ABB RobotStudio station: ProyectoLab.rsstn

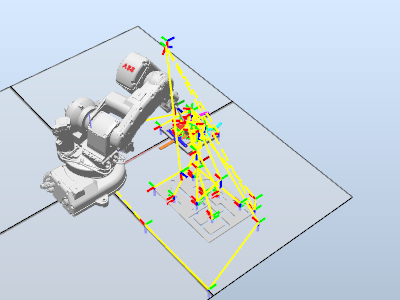
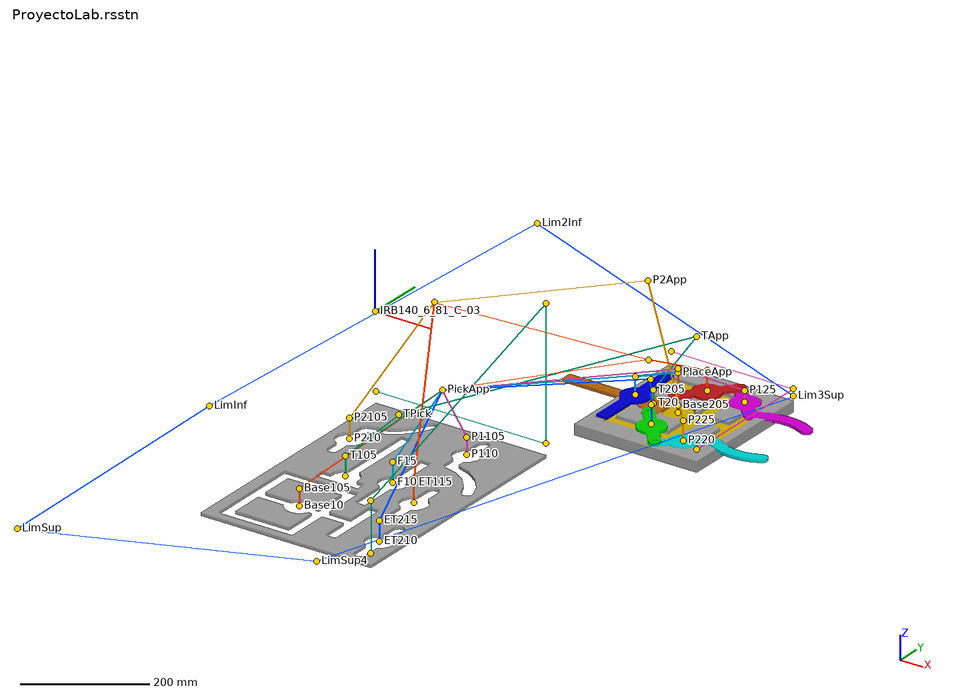
[picture v1: parts stored in the station drawn from their meshes, with robot base, taught points and paths (robot models come from the ABB library and are not in the file)]
Station ProyectoLab (saved by RobotStudio 22.2.9947.0)
Controller ProyectoLab
  mechanical unit ROB_1: IRB140_6_81_C_03, 6 joints, base frame (0, 0, 0) mm
Layout (positions relative to the parent item):
  - IRB140_6_81_C_03 [mechanism, from Robots\IRB140_6_81_C_G_03.rslib] at (0, 0, 0) mm; joint values [0.2279, 1.2634, -0.2779, 1.7688, -1.7005, -0.5808] (rad or m)
  - NewChupa [mechanism] at (606.41, 75.75, 144.2) mm, rotated rx -90 ry 89.52 rz 179.52 deg
      TCP NewChupa at (-10.65, -116.78, 115.87) mm, rotated rx -90 ry 89.52 rz -179.52 deg
      links: Chupita2
  - PiezaACortarApoyoInicialV3_0 [part] at (541.15, -381.68, 0) mm, rotated rx 90 ry 0 rz 180 deg, size 320 x 5 x 470 mm
  - TablaDejarV3 [part] at (639.18, -60.56, -43.75) mm, rotated rx 90 ry 0 rz 180 deg, size 230 x 19 x 260 mm
  - BaseGripper [part] at (583.77, -50.6, 10) mm, rotated rx 90 ry 0 rz 180 deg, size 200 x 5 x 180 mm
  - EslabonTransmisor1 [part] at (606.72, 23.71, 20) mm, rotated rx 90 ry 0 rz -39.33 deg, size 50 x 5 x 124.5 mm
  - EslabonTransmisor2 [part] at (606.64, -124.82, 20) mm, rotated rx 90 ry 0 rz 40 deg, size 50 x 5 x 124.5 mm
  - Pinza1 [part] at (672.04, 32.31, 20) mm, rotated rx -90 ry 0 rz 45 deg, size 111 x 5 x 174 mm
  - Pinza2 [part] at (672.04, -133.51, 15) mm, rotated rx 90 ry 0 rz -45 deg, size 111 x 5 x 174 mm
  - PlacaRetencion [part] at (523.76, -50.61, 20) mm, rotated rx 90 ry 0 rz 0 deg, size 49.7 x 5 x 180 mm
  - T [part] at (573.29, -50.6, 15) mm, rotated rx 90 ry 0 rz 180 deg, size 190 x 5 x 80 mm
  - IniB [smart component, from Components\Positioner.rslib]
      properties: Object=BaseGripper; Position=[0.28101 -0.63451 0]; Orientation=[1.5707963267949 0 3.14159265358979]; Reference=Global; ReferenceObject=(none)
  - IniT [smart component, from Components\Positioner.rslib]
      properties: Object=T; Position=[0.29968 -0.52272 0]; Orientation=[1.5707963267949 0 1.5707963267949]; Reference=Global; ReferenceObject=(none)
  - IniP1 [smart component, from Components\Positioner.rslib]
      properties: Object=Pinza1; Position=[0.40971 -0.3395 0.005]; Orientation=[-1.5707963267949 0 0]; Reference=Global; ReferenceObject=(none)
  - IniP2 [smart component, from Components\Positioner.rslib]
      properties: Object=Pinza2; Position=[0.2292 -0.39631 0]; Orientation=[1.5707963267949 0 0]; Reference=Global; ReferenceObject=(none)
  - IniE1 [smart component, from Components\Positioner.rslib]
      properties: Object=EslabonTransmisor1; Position=[0.43971 -0.52448 0]; Orientation=[1.5707963267949 0 0]; Reference=Global; ReferenceObject=(none)
  - IniE2 [smart component, from Components\Positioner.rslib]
      properties: Object=EslabonTransmisor2; Position=[0.47319 -0.6645 0]; Orientation=[1.5707963267949 0 0]; Reference=Global; ReferenceObject=(none)
  - IniPR [smart component, from Components\Positioner.rslib]
      properties: Object=PlacaRetencion; Position=[0.37233 -0.48425 0]; Orientation=[1.5707963267949 0 0]; Reference=Global; ReferenceObject=(none)
  - finB [smart component, from Components\Positioner.rslib]
      properties: Object=BaseGripper; Position=[0.58377 -0.0506 0.01]; Orientation=[1.5707963267949 0 -3.14159265358979]; Reference=Global; ReferenceObject=(none)
  - finT [smart component, from Components\Positioner.rslib]
      properties: Object=T; Position=[0.57329 -0.0506 0.015]; Orientation=[1.5707963267949 0 3.14159265358979]; Reference=Global; ReferenceObject=(none)
  - finP1 [smart component, from Components\Positioner.rslib]
      properties: Object=Pinza1; Position=[0.67204 0.03231 0.02]; Orientation=[-1.5707963267949 0 0.785398163397448]; Reference=Global; ReferenceObject=(none)
  - finP2 [smart component, from Components\Positioner.rslib]
      properties: Object=Pinza2; Position=[0.67204 -0.13351 0.015]; Orientation=[1.5707963267949 0 -0.785398163397448]; Reference=Global; ReferenceObject=(none)
  - finE1 [smart component, from Components\Positioner.rslib]
      properties: Object=EslabonTransmisor1; Position=[0.60672 0.02371 0.02]; Orientation=[1.5707963267949 0 -0.68643799480937]; Reference=Global; ReferenceObject=(none)
  - finE2 [smart component, from Components\Positioner.rslib]
      properties: Object=EslabonTransmisor2; Position=[0.60664 -0.12482 0.02]; Orientation=[1.5707963267949 0 0.698131700797732]; Reference=Global; ReferenceObject=(none)
  - finPR [smart component, from Components\Positioner.rslib]
      properties: Object=PlacaRetencion; Position=[0.52376 -0.05061 0.02]; Orientation=[1.5707963267949 0 0]; Reference=Global; ReferenceObject=(none)
  - Frame_1 [frame] at (127.2, 0.49, 126.37) mm, rotated rx -90 ry 89.52 rz -89.52 deg
Attachment: NewChupa is attached to IRB140_6_81_C_03 / Link6
Station signals: DI B1, DI B2, DI T1, DI T2, DI P11, DI P12, DI P21, DI P22, DI E11, DI E12, DI E21, DI E22, DI F1, DI F2
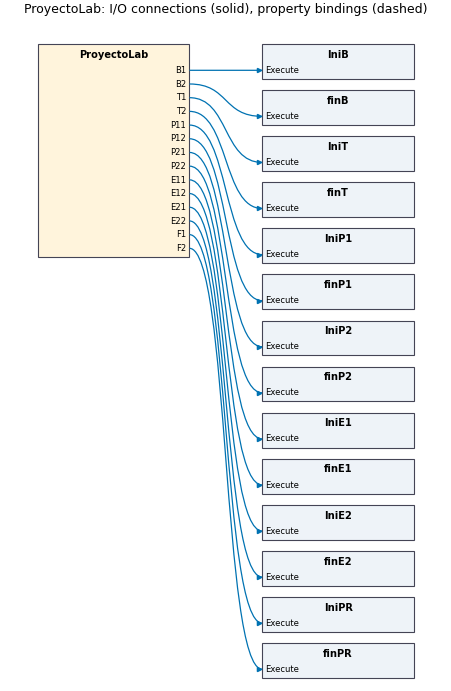
Station logic (signal -> signal, property => property):
  ProyectoLab.B1 -> IniB.Execute
  ProyectoLab.B2 -> finB.Execute
  ProyectoLab.T1 -> IniT.Execute
  ProyectoLab.T2 -> finT.Execute
  ProyectoLab.P11 -> IniP1.Execute
  ProyectoLab.P12 -> finP1.Execute
  ProyectoLab.P21 -> IniP2.Execute
  ProyectoLab.P22 -> finP2.Execute
  ProyectoLab.E11 -> IniE1.Execute
  ProyectoLab.E12 -> finE1.Execute
  ProyectoLab.E21 -> IniE2.Execute
  ProyectoLab.E22 -> finE2.Execute
  ProyectoLab.F1 -> IniPR.Execute
  ProyectoLab.F2 -> finPR.Execute
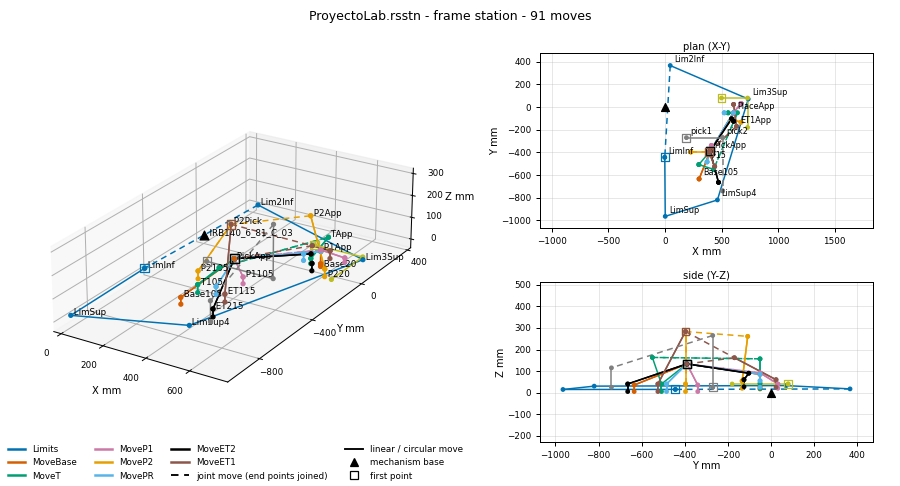
[picture p0: tool path of ProyectoLab.rsstn in frame station, 91 of 98 moves have a stored position in this frame; points joined in program order, loops and branches not executed]
Targets, tools, work objects and paths stored in the station, written as RAPID:
! task T_ROB1
MODULE CalibData
  PERS tooldata NewChupa:=[TRUE,[[127.2,0.485,126.368],[0.707106781,-0.005923775,0.707081968,0]],[1,[83.322,0.242,104.5],[1,0,0,0],0,0,0]];
  TASK PERS wobjdata World:=[FALSE,TRUE,"",[[0,0,0],[1,0,0,0]],[[0,0,0],[1,0,0,0]]];
  TASK PERS wobjdata NewPick:=[FALSE,TRUE,"",[[510,-270,5],[0,1,0,0]],[[0,0,0],[1,0,0,0]]];
  TASK PERS wobjdata NewPlace:=[FALSE,TRUE,"",[[730,80,20],[0,1,0,0]],[[0,0,0],[1,0,0,0]]];
ENDMODULE

! task T_ROB1
MODULE Module1
  CONST robtarget LimInf:=[[-1.268558474,-443.594527115,14.946918722],[0,0.707106781,0.707106781,0],[-1,-2,1,0],[9E+09,9E+09,9E+09,9E+09,9E+09,9E+09]];
  CONST robtarget LimSup:=[[2.920655475,-964.874814922,14.510384672],[0,0.707106781,0.707106781,0],[-1,-2,1,0],[9E+09,9E+09,9E+09,9E+09,9E+09,9E+09]];
  CONST robtarget LimSup4:=[[463.722752628,-820,30.05181616],[0,0.707106781,0.707106781,0],[-1,-2,1,0],[9E+09,9E+09,9E+09,9E+09,9E+09,9E+09]];
  CONST robtarget Lim3Sup:=[[735.880314711,71.133179396,32.548470254],[-0.000000014,0.707106783,0.707106779,0.000000019],[0,-1,1,0],[9E+09,9E+09,9E+09,9E+09,9E+09,9E+09]];
  CONST robtarget Lim2Inf:=[[46.954799307,367.02539237,17.249386066],[0,0.707106781,0.707106781,0],[0,-1,1,0],[9E+09,9E+09,9E+09,9E+09,9E+09,9E+09]];
  CONST robtarget PickApp:=[[-110.342872773,120.113138802,-128.175841477],[0.707106781,0,0,-0.707106781],[-1,0,-1,1],[9E+09,9E+09,9E+09,9E+09,9E+09,9E+09]];
  CONST robtarget Base105:=[[-207.99,364.51,-30],[0.707106781,0,0,-0.707106781],[-1,0,-1,1],[9E+09,9E+09,9E+09,9E+09,9E+09,9E+09]];
  CONST robtarget Base10:=[[-207.99,364.511,0],[0.707106781,0,0,-0.707106781],[-1,0,-1,1],[9E+09,9E+09,9E+09,9E+09,9E+09,9E+09]];
  CONST robtarget PlaceApp:=[[-125.227,130.603,-65],[0.707106781,0,0,-0.707106781],[0,1,-1,1],[9E+09,9E+09,9E+09,9E+09,9E+09,9E+09]];
  CONST robtarget Base205:=[[-125.227,130.604,-8.971],[0.707106781,0,0,-0.707106781],[0,1,-1,1],[9E+09,9E+09,9E+09,9E+09,9E+09,9E+09]];
  CONST robtarget Base20:=[[-125.227,130.604,3],[0.707106781,0,0,-0.707106781],[0,1,-1,1],[9E+09,9E+09,9E+09,9E+09,9E+09,9E+09]];
  CONST robtarget T105:=[[-210.324,237.721,-35],[0.707106781,0,0,-0.707106781],[-1,0,-1,1],[9E+09,9E+09,9E+09,9E+09,9E+09,9E+09]];
  CONST robtarget T10:=[[-210.324,237.721,0],[0.707106781,0,0,-0.707106781],[-1,0,-1,1],[9E+09,9E+09,9E+09,9E+09,9E+09,9E+09]];
  CONST robtarget TPick:=[[-80.342872773,280.113138802,-158.175841477],[0.707106781,0,0,-0.707106781],[-1,0,-1,1],[9E+09,9E+09,9E+09,9E+09,9E+09,9E+09]];
  CONST robtarget TApp:=[[-90.227,130.604,-136.705],[0,0,0,1],[-1,-1,0,1],[9E+09,9E+09,9E+09,9E+09,9E+09,9E+09]];
  CONST robtarget T205:=[[-171.711,130.604,-22.457885204],[0,0,0,1],[-1,-1,-1,1],[9E+09,9E+09,9E+09,9E+09,9E+09,9E+09]];
  CONST robtarget T20:=[[-171.711,130.604,1],[0,0,0,1],[-1,-1,-1,1],[9E+09,9E+09,9E+09,9E+09,9E+09,9E+09]];
  CONST robtarget P1105:=[[-100.292,69.504,-30],[0.707106781,0,0,-0.707106781],[-1,0,-1,1],[9E+09,9E+09,9E+09,9E+09,9E+09,9E+09]];
  CONST robtarget P110:=[[-100.292,69.504,0],[0.707106781,0,0,-0.707106781],[-1,0,-1,1],[9E+09,9E+09,9E+09,9E+09,9E+09,9E+09]];
  CONST robtarget P1App:=[[-125.227,130.604,-71.705],[0.382683433,0,0,-0.923879532],[0,0,-1,1],[9E+09,9E+09,9E+09,9E+09,9E+09,9E+09]];
  CONST robtarget P125:=[[-57.955,47.693,-20],[0.382683433,0,0,-0.923879532],[0,0,-1,1],[9E+09,9E+09,9E+09,9E+09,9E+09,9E+09]];
  CONST robtarget P120:=[[-57.955,47.693,0],[0.382683433,0,0,-0.923879532],[0,0,-1,1],[9E+09,9E+09,9E+09,9E+09,9E+09,9E+09]];
  CONST robtarget P2Pick:=[[-121.178397921,126.307,-278.381942838],[0,0,0,1],[-1,1,-2,0],[9E+09,9E+09,9E+09,9E+09,9E+09,9E+09]];
  CONST robtarget P2105:=[[-280.797,126.307,-35],[0,0,0,1],[-1,1,-2,0],[9E+09,9E+09,9E+09,9E+09,9E+09,9E+09]];
  CONST robtarget P210:=[[-280.797,126.307,0],[0,0,0,1],[-1,1,-2,0],[9E+09,9E+09,9E+09,9E+09,9E+09,9E+09]];
  CONST robtarget P2App:=[[-142.214371526,187.704774603,-240.969916699],[0.382683433,0,0,-0.923879532],[0,0,-1,1],[9E+09,9E+09,9E+09,9E+09,9E+09,9E+09]];
  CONST robtarget P225:=[[-57.864,213.606,-34.204],[0.382683433,0,0,-0.923879532],[0,0,-1,1],[9E+09,9E+09,9E+09,9E+09,9E+09,9E+09]];
  CONST robtarget P220:=[[-57.864,213.606,0],[0.382683432,0,0,-0.923879533],[0,0,-1,1],[9E+09,9E+09,9E+09,9E+09,9E+09,9E+09]];
  CONST robtarget F15:=[[-137.666,214.247,-35],[0.707106781,0,0,-0.707106781],[-1,0,-1,1],[9E+09,9E+09,9E+09,9E+09,9E+09,9E+09]];
  CONST robtarget F10:=[[-137.666,214.247,0],[0.707106781,0,0,-0.707106781],[-1,0,-1,1],[9E+09,9E+09,9E+09,9E+09,9E+09,9E+09]];
  CONST robtarget F25:=[[-206.227,130.603,-35],[0.707106781,0,0,-0.707106781],[0,1,-1,1],[9E+09,9E+09,9E+09,9E+09,9E+09,9E+09]];
  CONST robtarget F20:=[[-206.227,130.603,-5],[0.707106781,0,0,-0.707106781],[0,1,-1,1],[9E+09,9E+09,9E+09,9E+09,9E+09,9E+09]];
  CONST robtarget ET215:=[[-36.814,394.504,-35],[0.707106781,0,0,-0.707106781],[-1,0,-1,1],[9E+09,9E+09,9E+09,9E+09,9E+09,9E+09]];
  CONST robtarget ET210:=[[-36.814,394.504,0],[0.707106781,0,0,-0.707106781],[-1,0,-1,1],[9E+09,9E+09,9E+09,9E+09,9E+09,9E+09]];
  CONST robtarget ET2App:=[[-141.14536065,182.779436275,-69.962726226],[0.382683433,0,0,-0.923879532],[0,0,-1,1],[9E+09,9E+09,9E+09,9E+09,9E+09,9E+09]];
  CONST robtarget ET225:=[[-123.166,204.988,-40],[0.422618262,0,0,-0.906307787],[0,0,-1,1],[9E+09,9E+09,9E+09,9E+09,9E+09,9E+09]];
  CONST robtarget ET220:=[[-123.36,204.834,-7.096],[0.422618262,0,0,-0.906307787],[0,0,-1,1],[9E+09,9E+09,9E+09,9E+09,9E+09,9E+09]];
  CONST robtarget ET115:=[[-70.294,254.478,-35],[0,0,0,1],[-1,1,-2,0],[9E+09,9E+09,9E+09,9E+09,9E+09,9E+09]];
  CONST robtarget ET110:=[[-70.293,254.479,0],[0,0,0,1],[-1,1,-2,0],[9E+09,9E+09,9E+09,9E+09,9E+09,9E+09]];
  CONST robtarget ET1App:=[[-97.458484126,249.43301943,-141.897823694],[0.336487213,0,0,-0.941688035],[-1,0,-1,1],[9E+09,9E+09,9E+09,9E+09,9E+09,9E+09]];
  CONST robtarget ET125:=[[-123.284,56.288,-40],[0.336487213,0,0,-0.941688035],[0,0,-1,1],[9E+09,9E+09,9E+09,9E+09,9E+09,9E+09]];
  CONST robtarget ET120:=[[-123.284,56.288,-5],[0.336487213,0,0,-0.941688035],[0,0,-1,1],[9E+09,9E+09,9E+09,9E+09,9E+09,9E+09]];
  CONST jointtarget Home:=[[0,0,0,0,30,0],[9E+09,9E+09,9E+09,9E+09,9E+09,9E+09]];
  CONST jointtarget tool:=[[-89.3,42.5,-51.4,0,0,0],[9E+09,9E+09,9E+09,9E+09,9E+09,9E+09]];
  CONST robtarget pick1:=[[190,-270,25],[0,0,1,0],[-2,1,1,0],[9E+09,9E+09,9E+09,9E+09,9E+09,9E+09]];
  CONST robtarget pick2:=[[510,-270,25],[0,0,1,0],[-1,1,2,0],[9E+09,9E+09,9E+09,9E+09,9E+09,9E+09]];
  CONST robtarget pick25:=[[510,-270,265],[0,0,1,0],[-1,1,2,0],[9E+09,9E+09,9E+09,9E+09,9E+09,9E+09]];
  CONST robtarget pick35:=[[510,-740,115],[0,0.707106781,0.707106781,0],[-1,-2,1,0],[9E+09,9E+09,9E+09,9E+09,9E+09,9E+09]];
  CONST robtarget pick3:=[[510,-740,25],[0,0.707106781,0.707106781,0],[-1,-2,1,0],[9E+09,9E+09,9E+09,9E+09,9E+09,9E+09]];
  CONST robtarget place1:=[[500,80,40],[0,0,1,0],[0,-2,-2,0],[9E+09,9E+09,9E+09,9E+09,9E+09,9E+09]];
  CONST robtarget place2:=[[730,80,40],[0,0,1,0],[0,-2,-3,0],[9E+09,9E+09,9E+09,9E+09,9E+09,9E+09]];
  CONST robtarget place3:=[[730,-180,40],[0,0,1,0],[-1,-3,-2,0],[9E+09,9E+09,9E+09,9E+09,9E+09,9E+09]];
  CONST jointtarget HomeFinal:=[[0,0,0,0,0,0],[9E+09,9E+09,9E+09,9E+09,9E+09,9E+09]];
  PROC main()
    Homing;
    Set DO_03;
    WaitDI DI_01,1;
    DefinePick;
    WaitDI DI_01,1;
    DefinePlace;
    WaitDI DI_01,1;
    MoveBase;
    WaitDI DI_01,1;
    MoveT;
    WaitDI DI_01,1;
    MoveP1;
    WaitDI DI_01,1;
    MoveP2;
    WaitDI DI_01,1;
    MoveET1;
    WaitDI DI_01,1;
    MoveET2;
    WaitDI DI_01,1;
    MovePR;
    WaitDI DI_01,1;
    Final;
    Reset DO_03;
  ENDPROC
  PROC Limits()
    MoveJ LimInf,v150,fine,NewChupa\WObj:=World;
    MoveL LimSup,v150,fine,NewChupa\WObj:=World;
    MoveL LimSup4,v150,fine,NewChupa\WObj:=World;
    MoveL Lim3Sup,v150,fine,NewChupa\WObj:=World;
    MoveL Lim2Inf,v150,fine,NewChupa\WObj:=World;
    MoveJ LimInf,v150,fine,NewChupa\WObj:=World;
  ENDPROC
  PROC MoveBase()
    MoveJ PickApp,v100,fine,NewChupa\WObj:=NewPick;
    MoveJ PickApp,v100,fine,NewChupa\WObj:=NewPick;
    MoveL Base105,v100,fine,NewChupa\WObj:=NewPick;
    MoveLDO Base10,v50,fine,NewChupa\WObj:=NewPick,DO_01,1;
    Set DO_01;
    WaitTime 3;
    Reset DO_01;
    MoveL Base105,v50,fine,NewChupa\WObj:=NewPick;
    MoveL PickApp,v100,fine,NewChupa\WObj:=NewPick;
    MoveL PlaceApp,v100,fine,NewChupa\WObj:=NewPlace;
    MoveL Base205,v100,fine,NewChupa\WObj:=NewPlace;
    WaitDI DI_01,1;
    MoveLDO Base20,v50,fine,NewChupa\WObj:=NewPlace,DO_02,1;
    Set DO_02;
    WaitTime 3;
    Reset DO_02;
    MoveL Base205,v50,fine,NewChupa\WObj:=NewPlace;
    MoveL PlaceApp,v100,fine,NewChupa\WObj:=NewPlace;
    MoveL PickApp,v100,fine,NewChupa\WObj:=NewPick;
  ENDPROC
  PROC MoveT()
    MoveJ PickApp,v100,fine,NewChupa\WObj:=NewPick;
    MoveL T105,v100,fine,NewChupa\WObj:=NewPick;
    MoveLDO T10,v50,fine,NewChupa\WObj:=NewPick,DO_01,1;
    Set DO_01;
    WaitTime 3;
    Reset DO_01;
    MoveL T105,v100,fine,NewChupa\WObj:=NewPick;
    MoveL TPick,v100,fine,NewChupa\WObj:=NewPick;
    MoveJ TApp,v100,fine,NewChupa\WObj:=NewPlace;
    MoveL T205,v100,fine,NewChupa\WObj:=NewPlace;
    WaitDI DI_01,1;
    MoveLDO T20,v50,fine,NewChupa\WObj:=NewPlace,DO_02,1;
    Set DO_02;
    WaitTime 3;
    Reset DO_02;
    MoveL T205,v100,fine,NewChupa\WObj:=NewPlace;
    MoveL TApp,v100,fine,NewChupa\WObj:=NewPlace;
    MoveJ TPick,v100,fine,NewChupa\WObj:=NewPick;
  ENDPROC
  PROC MoveP1()
    MoveJ PickApp,v100,fine,NewChupa\WObj:=NewPick;
    MoveL P1105,v100,fine,NewChupa\WObj:=NewPick;
    MoveLDO P110,v50,fine,NewChupa\WObj:=NewPick,DO_01,1;
    Set DO_01;
    WaitTime 3;
    Reset DO_01;
    MoveL P1105,v100,fine,NewChupa\WObj:=NewPick;
    MoveL PickApp,v100,fine,NewChupa\WObj:=NewPick;
    MoveJ P1App,v100,fine,NewChupa\WObj:=NewPlace;
    MoveL P125,v100,fine,NewChupa\WObj:=NewPlace;
    WaitDI DI_01,1;
    MoveLDO P120,v50,fine,NewChupa\WObj:=NewPlace,DO_02,1;
    Set DO_02;
    WaitTime 3;
    Reset DO_02;
    MoveL P125,v100,fine,NewChupa\WObj:=NewPlace;
    MoveL P1App,v100,fine,NewChupa\WObj:=NewPlace;
    MoveJ PickApp,v100,fine,NewChupa\WObj:=NewPick;
  ENDPROC
  PROC MoveP2()
    MoveJ P2Pick,v100,fine,NewChupa\WObj:=NewPick;
    MoveL P2105,v100,fine,NewChupa\WObj:=NewPick;
    MoveLDO P210,v50,fine,NewChupa\WObj:=NewPick,DO_01,1;
    Set DO_01;
    WaitTime 3;
    Reset DO_01;
    MoveL P2105,v100,fine,NewChupa\WObj:=NewPick;
    MoveJ P2Pick,v100,fine,NewChupa\WObj:=NewPick;
    MoveJ P2App,v100,fine,NewChupa\WObj:=NewPlace;
    MoveL P225,v100,fine,NewChupa\WObj:=NewPlace;
    WaitDI DI_01,1;
    MoveLDO P220,v50,fine,NewChupa\WObj:=NewPlace,DO_02,1;
    Set DO_02;
    WaitTime 3;
    Reset DO_02;
    MoveL P225,v100,fine,NewChupa\WObj:=NewPlace;
    MoveL P2App,v100,fine,NewChupa\WObj:=NewPlace;
  ENDPROC
  PROC MovePR()
    MoveJ PickApp,v100,fine,NewChupa\WObj:=NewPick;
    MoveL F15,v100,fine,NewChupa\WObj:=NewPick;
    MoveLDO F10,v50,fine,NewChupa\WObj:=NewPick,DO_01,1;
    Set DO_01;
    WaitTime 3;
    Reset DO_01;
    MoveL F15,v50,fine,NewChupa\WObj:=NewPick;
    MoveL PickApp,v100,fine,NewChupa\WObj:=NewPick;
    MoveL PlaceApp,v100,fine,NewChupa\WObj:=NewPlace;
    MoveL F25,v100,fine,NewChupa\WObj:=NewPlace;
    WaitDI DI_01,1;
    MoveLDO F20,v50,fine,NewChupa\WObj:=NewPlace,DO_02,1;
    Set DO_02;
    WaitTime 3;
    Reset DO_02;
    MoveL F25,v50,fine,NewChupa\WObj:=NewPlace;
    MoveL PlaceApp,v100,fine,NewChupa\WObj:=NewPlace;
    MoveL PickApp,v100,fine,NewChupa\WObj:=NewPick;
  ENDPROC
  PROC MoveET2()
    MoveJ PickApp,v100,fine,NewChupa\WObj:=NewPick;
    MoveL ET215,v100,fine,NewChupa\WObj:=NewPick;
    MoveLDO ET210,v50,fine,NewChupa\WObj:=NewPick,DO_01,1;
    Set DO_01;
    WaitTime 3;
    Reset DO_01;
    MoveL ET215,v50,fine,NewChupa\WObj:=NewPick;
    MoveL PickApp,v100,fine,NewChupa\WObj:=NewPick;
    MoveL ET2App,v100,fine,NewChupa\WObj:=NewPlace;
    MoveL ET225,v50,fine,NewChupa\WObj:=NewPlace;
    WaitDI DI_01,1;
    MoveLDO ET220,v50,fine,NewChupa\WObj:=NewPlace,DO_02,1;
    Set DO_02;
    WaitTime 3;
    Reset DO_02;
    MoveL ET225,v50,fine,NewChupa\WObj:=NewPlace;
    MoveL ET2App,v100,fine,NewChupa\WObj:=NewPlace;
    MoveL PickApp,v100,fine,NewChupa\WObj:=NewPick;
  ENDPROC
  PROC MoveET1()
    MoveJ P2Pick,v100,fine,NewChupa\WObj:=NewPick;
    MoveL ET115,v100,fine,NewChupa\WObj:=NewPick;
    MoveLDO ET110,v50,fine,NewChupa\WObj:=NewPick,DO_01,1;
    Set DO_01;
    WaitTime 3;
    Reset DO_01;
    MoveL ET115,v100,fine,NewChupa\WObj:=NewPick;
    MoveL P2Pick,v100,fine,NewChupa\WObj:=NewPick;
    MoveJ ET1App,v100,fine,NewChupa\WObj:=NewPlace;
    MoveL ET125,v100,fine,NewChupa\WObj:=NewPlace;
    WaitDI DI_01,1;
    MoveLDO ET120,v50,fine,NewChupa\WObj:=NewPlace,DO_02,1;
    Set DO_02;
    WaitTime 3;
    Reset DO_02;
    MoveL ET125,v100,fine,NewChupa\WObj:=NewPlace;
    MoveL ET1App,v100,fine,NewChupa\WObj:=NewPlace;
    MoveJ PickApp,v100,fine,NewChupa\WObj:=NewPick;
  ENDPROC
  PROC Homing()
    MoveAbsJ Home,v200,fine,NewChupa\WObj:=NewPlace;
  ENDPROC
  PROC ToolSet()
    MoveAbsJ Home,v300,fine,NewChupa\WObj:=wobj0;
    WaitDI DI_01,1;
    MoveAbsJ tool,v300,fine,NewChupa\WObj:=wobj0;
    WaitDI DI_01,1;
    MoveAbsJ Home,v300,fine,NewChupa\WObj:=wobj0;
  ENDPROC
  PROC DefinePick()
    MoveJ pick1,v300,fine,NewChupa\WObj:=World;
    WaitDI DI_01,1;
    MoveL pick2,v300,fine,NewChupa\WObj:=World;
    WaitDI DI_01,1;
    MoveL pick25,v300,fine,NewChupa\WObj:=World;
    MoveJ pick35,v300,fine,NewChupa\WObj:=World;
    MoveL pick3,v300,fine,NewChupa\WObj:=World;
    WaitDI DI_01,1;
    MoveAbsJ Home,v300,fine,NewChupa\WObj:=wobj0;
  ENDPROC
  PROC DefinePlace()
    MoveJ place1,v300,fine,NewChupa\WObj:=World;
    WaitDI DI_01,1;
    MoveL place2,v300,fine,NewChupa\WObj:=World;
    WaitDI DI_01,1;
    MoveL place3,v300,fine,NewChupa\WObj:=World;
    WaitDI DI_01,1;
    MoveAbsJ Home,v300,fine,NewChupa\WObj:=wobj0;
  ENDPROC
  PROC Final()
    MoveAbsJ HomeFinal,v300,fine,NewChupa\WObj:=NewPick;
  ENDPROC
ENDMODULE

